% RSLogix 500 project 4P4_E_with_comments.RSS, saved by version 8.30.00.16 %
PROJECT "4P4_E"    % processor: MicroLogix 1000 %

PROGRAM FILES
  LAD 2 "MAIN_PROG"  6 rungs
  LAD 3 "USER_FAULT"  2 rungs
  LAD 4 "HSC_INT"  1 rungs
  LAD 5 "STI_INT"  9 rungs
  LAD 7   40 rungs
  LAD 6, 8, 9, 10, 11, 12, 13, 14, 15, 16: only END

DATA FILES
  O0 OUTPUT  1 elements
  I1 INPUT  2 elements
  S2 STATUS  33 elements
  B3 BINARY  32 elements
  T4 TIMER  40 elements
  C5 COUNTER  32 elements
  R6 CONTROL  16 elements
  N7 INTEGER  105 elements

LADDER 2 "MAIN_PROG"
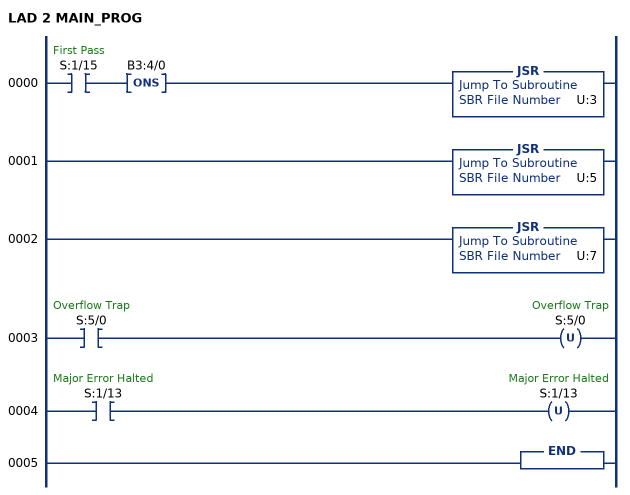
% Rung: 0 %
SOR XIC S:1/15 OSR B3:4/0 JSR U:3 EOR
%   S:1/15  "First Pass" %
% Rung: 1 %
SOR JSR U:5 EOR
% Rung: 2 %
SOR JSR U:7 EOR
% Rung: 3 %
SOR XIC S:5/0 OTU S:5/0 EOR
%   S:5/0  "Overflow Trap" %
% Rung: 4 %
SOR XIC S:1/13 OTU S:1/13 EOR
%   S:1/13  "Major Error Halted" %
% Rung: 5 %
SOR END EOR

LADDER 3 "USER_FAULT"
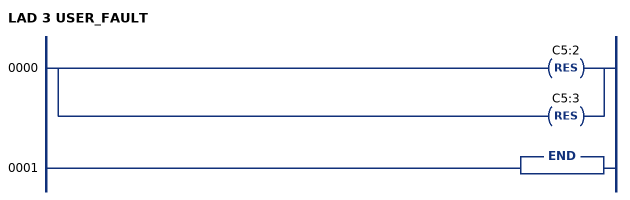
% Rung: 0 %
SOR BST RES C5:2 NXB RES C5:3 BND EOR
% Rung: 1 %
SOR END EOR

LADDER 5 "STI_INT"
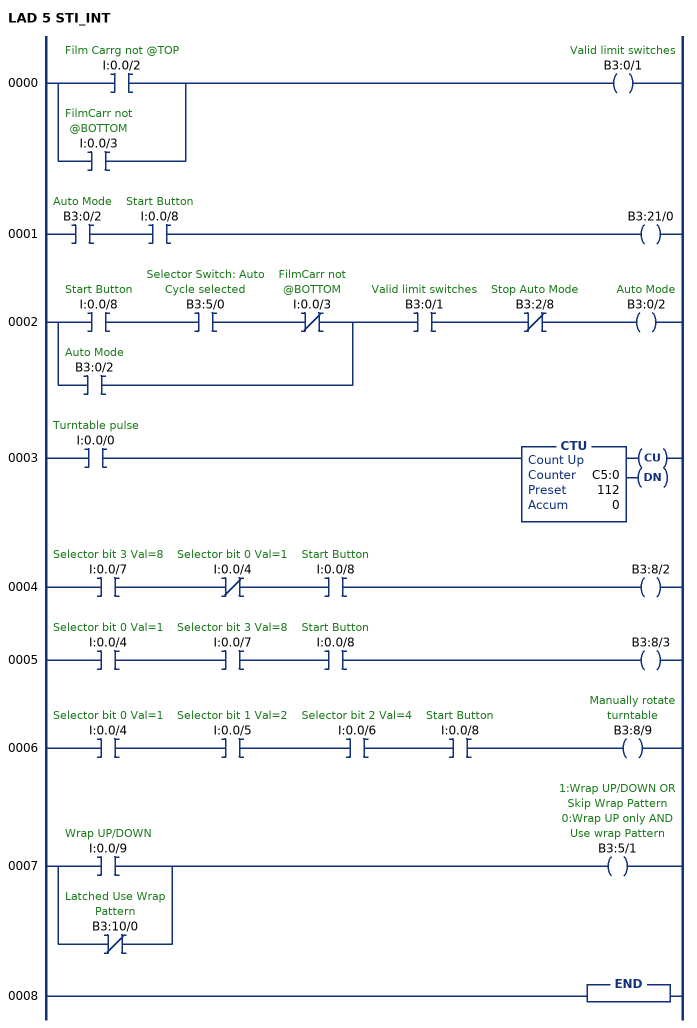
% Rung: 0 %
SOR BST XIC I:0.0/2 NXB XIC I:0.0/3 BND OTE B3:0/1 EOR
%   I:0.0/2  "Film Carrg not @TOP" %
%   XIC I:0.0/2  "1:Film Carr not @TOP" %
%   I:0.0/3  "FilmCarr not @BOTTOM" %
%   XIC I:0.0/3  "1:FilmCarr not@BOTTM" %
%   B3:0/1  "Valid limit switches" %
% Rung: 1 %
SOR XIC B3:0/2 XIC I:0.0/8 OTE B3:21/0 EOR
%   B3:0/2  "Auto Mode" %
%   XIC B3:0/2  "1:Auto" %
%   I:0.0/8  "Start Button" %
% Rung: 2 %
SOR BST XIC I:0.0/8 XIC B3:5/0 XIO I:0.0/3 NXB XIC B3:0/2 BND XIC B3:0/1 XIO B3:2/8 OTE B3:0/2 EOR
%   I:0.0/8  "Start Button" %
%   B3:5/0  "Selector Switch: Auto Cycle selected" %
%   I:0.0/3  "FilmCarr not @BOTTOM" %
%   XIO I:0.0/3  "0:Film Carrg @BOTTOM" %
%   B3:0/2  "Auto Mode" %
%   XIC B3:0/2  "1:Auto" %
%   B3:0/1  "Valid limit switches" %
%   B3:2/8  "Stop Auto Mode" %
%   XIO B3:2/8  "0:Continue Auto Mode" %
% Rung: 3 %
SOR XIC I:0.0/0 CTU C5:0 112 0 EOR
%   I:0.0/0  "Turntable pulse" %
%   XIC I:0.0/0  "1:Turntable pulse on" %
% Rung: 4 %
SOR XIC I:0.0/7 XIO I:0.0/4 XIC I:0.0/8 OTE B3:8/2 EOR
%   I:0.0/7  "Selector bit 3 Val=8" %
%   I:0.0/4  "Selector bit 0 Val=1" %
%   I:0.0/8  "Start Button" %
% Rung: 5 %
SOR XIC I:0.0/4 XIC I:0.0/7 XIC I:0.0/8 OTE B3:8/3 EOR
%   I:0.0/4  "Selector bit 0 Val=1" %
%   I:0.0/7  "Selector bit 3 Val=8" %
%   I:0.0/8  "Start Button" %
% Rung: 6 %
SOR XIC I:0.0/4 XIC I:0.0/5 XIC I:0.0/6 XIC I:0.0/8 OTE B3:8/9 EOR
%   I:0.0/4  "Selector bit 0 Val=1" %
%   I:0.0/5  "Selector bit 1 Val=2" %
%   I:0.0/6  "Selector bit 2 Val=4" %
%   I:0.0/8  "Start Button" %
%   B3:8/9  "Manually rotate turntable" %
% Rung: 7 %
SOR BST XIC I:0.0/9 NXB XIO B3:10/0 BND OTE B3:5/1 EOR
%   I:0.0/9  "Wrap UP/DOWN" %
%   B3:10/0  "Latched Use Wrap Pattern" %
%   XIO B3:10/0  "0:Skip Wrap Pattern" %
%   B3:5/1  "1:Wrap UP/DOWN OR Skip Wrap Pattern 0:Wrap UP only AND Use wrap Pattern" %
% Rung: 8 %
SOR END EOR

LADDER 7
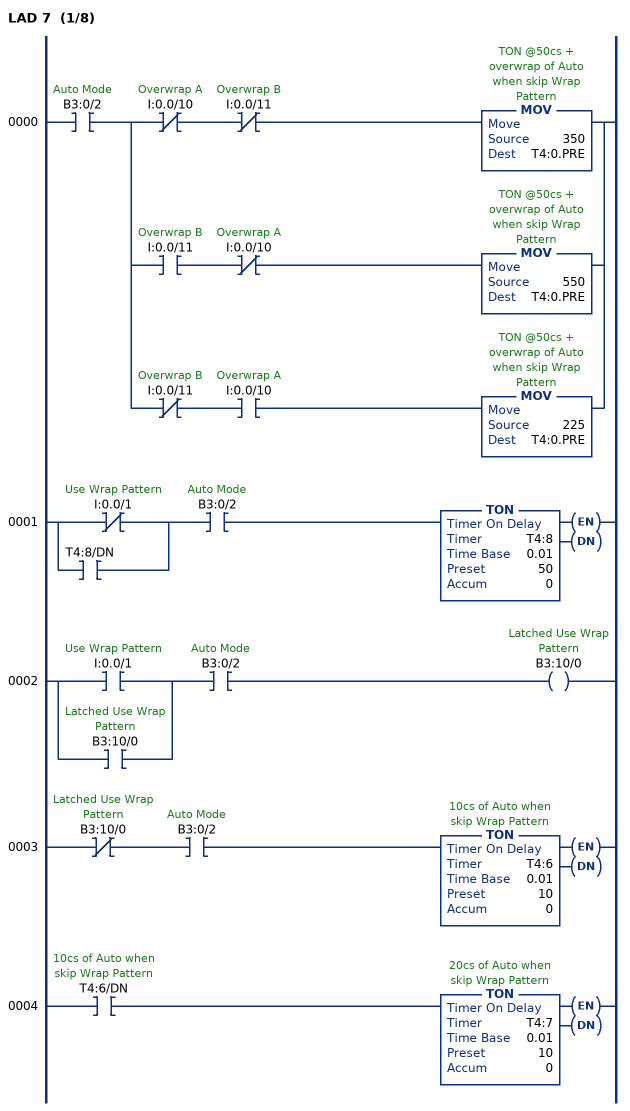
% Rung: 0 %
SOR XIC B3:0/2 BST XIO I:0.0/10 XIO I:0.0/11 MOV 350 T4:0.PRE NXB XIC I:0.0/11 XIO I:0.0/10 MOV 550 T4:0.PRE NXB XIO I:0.0/11 XIC I:0.0/10 MOV 225 T4:0.PRE BND EOR
%   B3:0/2  "Auto Mode" %
%   XIC B3:0/2  "1:Auto" %
%   I:0.0/10  "Overwrap A" %
%   I:0.0/11  "Overwrap B" %
%   T4:0  "TON @50cs + overwrap of Auto when skip Wrap Pattern" %
% Rung: 1 %
SOR BST XIO I:0.0/1 NXB XIC T4:8/DN BND XIC B3:0/2 TON T4:8 0.01 50 0 EOR
%   I:0.0/1  "Use Wrap Pattern" %
%   XIO I:0.0/1  "0:Skip Wrap Pattern => No UP/DOWN" %
%   B3:0/2  "Auto Mode" %
%   XIC B3:0/2  "1:Auto" %
% Rung: 2 %
SOR BST XIC I:0.0/1 NXB XIC B3:10/0 BND XIC B3:0/2 OTE B3:10/0 EOR
%   I:0.0/1  "Use Wrap Pattern" %
%   XIC I:0.0/1  "1:Use Wrap Pattern" %
%   B3:10/0  "Latched Use Wrap Pattern" %
%   B3:0/2  "Auto Mode" %
%   XIC B3:0/2  "1:Auto" %
% Rung: 3 %
SOR XIO B3:10/0 XIC B3:0/2 TON T4:6 0.01 10 0 EOR
%   B3:10/0  "Latched Use Wrap Pattern" %
%   XIO B3:10/0  "0:Skip Wrap Pattern" %
%   B3:0/2  "Auto Mode" %
%   XIC B3:0/2  "1:Auto" %
%   T4:6  "10cs of Auto when skip Wrap Pattern" %
% Rung: 4 %
SOR XIC T4:6/DN TON T4:7 0.01 10 0 EOR
%   T4:6  "10cs of Auto when skip Wrap Pattern" %
%   XIC T4:6/DN  "1:Bypass TOP band 1:10cs+ of Auto when skip Wrap Pattern" %
%   T4:7  "20cs of Auto when skip Wrap Pattern" %

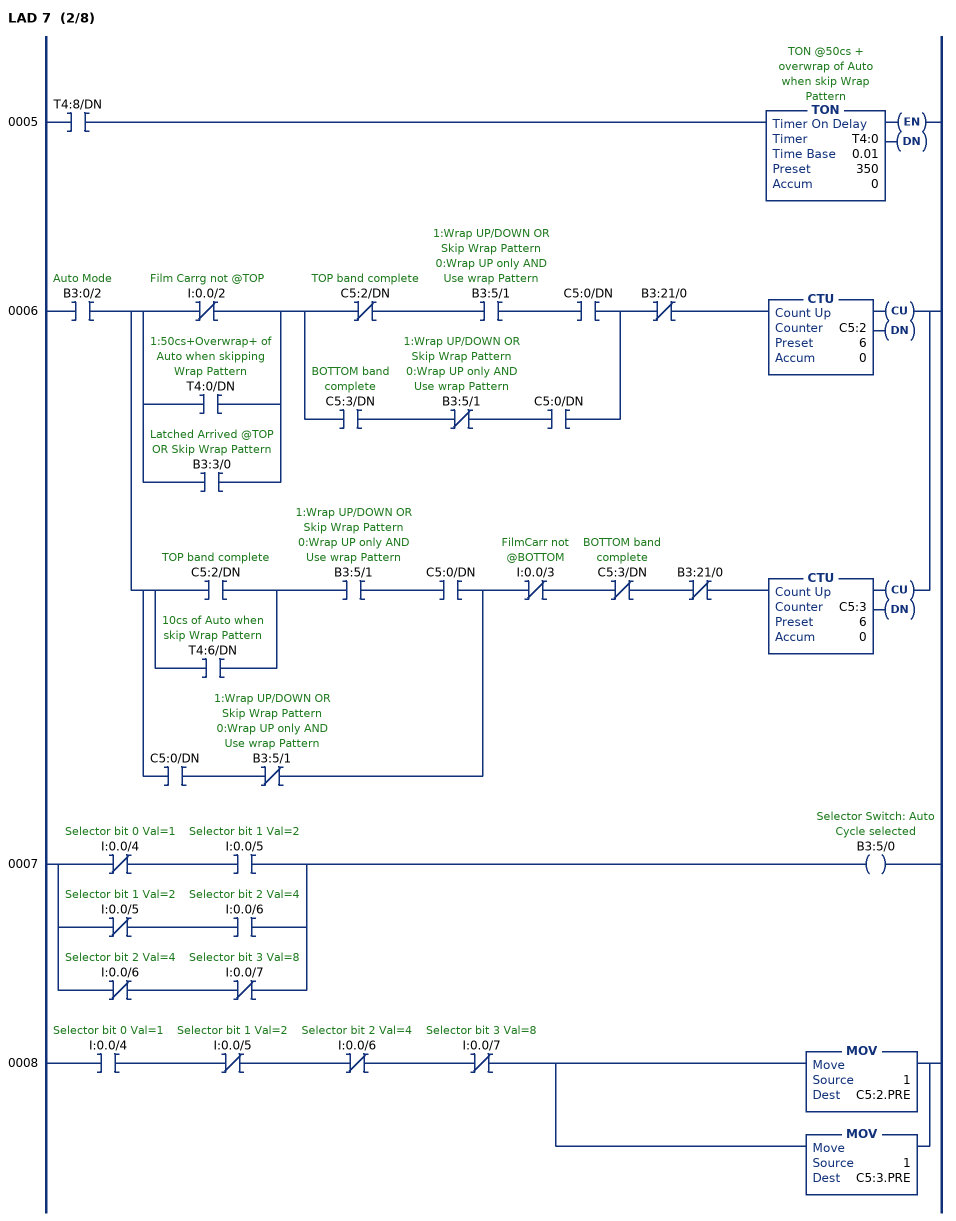
% Rung: 5 %
SOR XIC T4:8/DN TON T4:0 0.01 350 0 EOR
%   T4:0  "TON @50cs + overwrap of Auto when skip Wrap Pattern" %
% Rung: 6 %
SOR XIC B3:0/2 BST BST XIO I:0.0/2 NXB XIC T4:0/DN NXB XIC B3:3/0 BND BST XIO C5:2/DN XIC B3:5/1 XIC C5:0/DN NXB XIC C5:3/DN XIO B3:5/1 XIC C5:0/DN BND XIO B3:21/0 CTU C5:2 6 0 NXB BST BST XIC C5:2/DN NXB XIC T4:6/DN BND XIC B3:5/1 XIC C5:0/DN NXB XIC C5:0/DN XIO B3:5/1 BND XIO I:0.0/3 XIO C5:3/DN XIO B3:21/0 CTU C5:3 6 0 BND EOR
%   B3:0/2  "Auto Mode" %
%   XIC B3:0/2  "1:Auto" %
%   I:0.0/2  "Film Carrg not @TOP" %
%   XIO I:0.0/2  "0:Film Carriage @TOP" %
%   T4:0/DN  "1:50cs+Overwrap+ of Auto when skipping Wrap Pattern" %
%   B3:3/0  "Latched Arrived @TOP OR Skip Wrap Pattern" %
%   XIC B3:3/0  "1:Arrived @TOP OR Skip Wrap Pattern" %
%   C5:2/DN  "TOP band complete" %
%   B3:5/1  "1:Wrap UP/DOWN OR Skip Wrap Pattern 0:Wrap UP only AND Use wrap Pattern" %
%   XIC B3:5/1  "1:Bypass BOTTOM band 1:Wrap UP/DOWN OR Skip Wrap Pattern" %
%   C5:3/DN  "BOTTOM band complete" %
%   XIO B3:5/1  "0:Wrap UP only AND Use wrap Pattern" %
%   T4:6  "10cs of Auto when skip Wrap Pattern" %
%   XIC T4:6/DN  "1:Bypass TOP band 1:10cs+ of Auto when skip Wrap Pattern" %
%   I:0.0/3  "FilmCarr not @BOTTOM" %
%   XIO I:0.0/3  "0:Film Carrg @BOTTOM" %
% Rung: 7 %
SOR BST XIO I:0.0/4 XIC I:0.0/5 NXB XIO I:0.0/5 XIC I:0.0/6 NXB XIO I:0.0/6 XIO I:0.0/7 BND OTE B3:5/0 EOR
%   I:0.0/4  "Selector bit 0 Val=1" %
%   I:0.0/5  "Selector bit 1 Val=2" %
%   I:0.0/6  "Selector bit 2 Val=4" %
%   I:0.0/7  "Selector bit 3 Val=8" %
%   B3:5/0  "Selector Switch: Auto Cycle selected" %
% Rung: 8 %
SOR XIC I:0.0/4 XIO I:0.0/5 XIO I:0.0/6 XIO I:0.0/7 BST MOV 1 C5:2.PRE NXB MOV 1 C5:3.PRE BND EOR
%   I:0.0/4  "Selector bit 0 Val=1" %
%   I:0.0/5  "Selector bit 1 Val=2" %
%   I:0.0/6  "Selector bit 2 Val=4" %
%   I:0.0/7  "Selector bit 3 Val=8" %

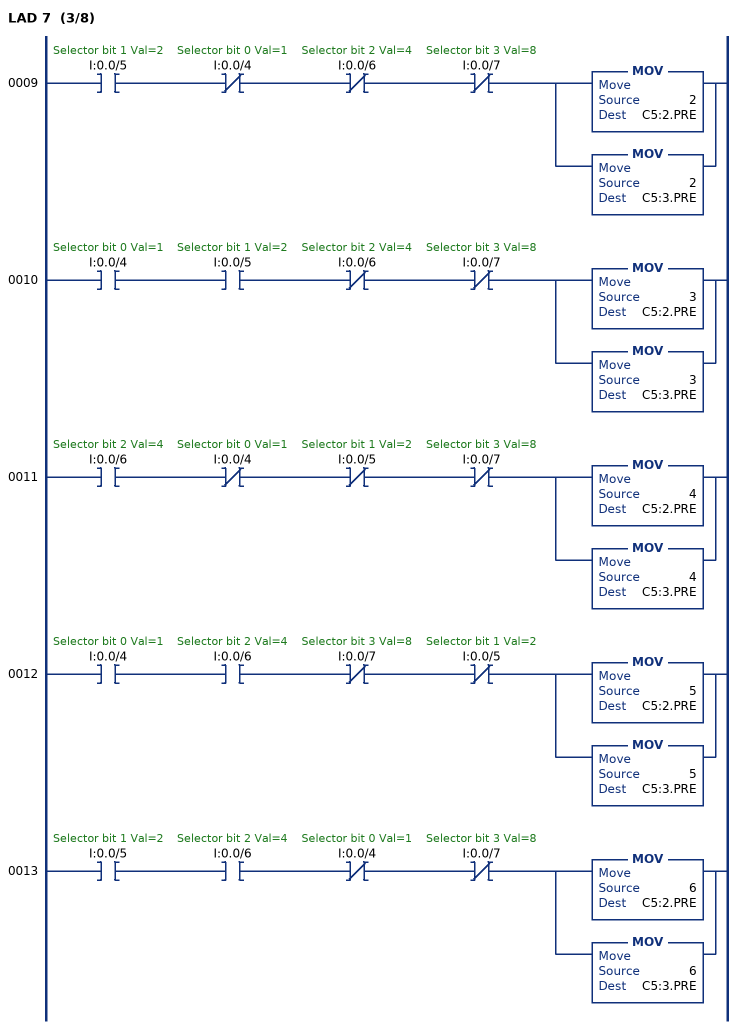
% Rung: 9 %
SOR XIC I:0.0/5 XIO I:0.0/4 XIO I:0.0/6 XIO I:0.0/7 BST MOV 2 C5:2.PRE NXB MOV 2 C5:3.PRE BND EOR
%   I:0.0/5  "Selector bit 1 Val=2" %
%   I:0.0/4  "Selector bit 0 Val=1" %
%   I:0.0/6  "Selector bit 2 Val=4" %
%   I:0.0/7  "Selector bit 3 Val=8" %
% Rung: 10 %
SOR XIC I:0.0/4 XIC I:0.0/5 XIO I:0.0/6 XIO I:0.0/7 BST MOV 3 C5:2.PRE NXB MOV 3 C5:3.PRE BND EOR
%   I:0.0/4  "Selector bit 0 Val=1" %
%   I:0.0/5  "Selector bit 1 Val=2" %
%   I:0.0/6  "Selector bit 2 Val=4" %
%   I:0.0/7  "Selector bit 3 Val=8" %
% Rung: 11 %
SOR XIC I:0.0/6 XIO I:0.0/4 XIO I:0.0/5 XIO I:0.0/7 BST MOV 4 C5:2.PRE NXB MOV 4 C5:3.PRE BND EOR
%   I:0.0/6  "Selector bit 2 Val=4" %
%   I:0.0/4  "Selector bit 0 Val=1" %
%   I:0.0/5  "Selector bit 1 Val=2" %
%   I:0.0/7  "Selector bit 3 Val=8" %
% Rung: 12 %
SOR XIC I:0.0/4 XIC I:0.0/6 XIO I:0.0/7 XIO I:0.0/5 BST MOV 5 C5:2.PRE NXB MOV 5 C5:3.PRE BND EOR
%   I:0.0/4  "Selector bit 0 Val=1" %
%   I:0.0/6  "Selector bit 2 Val=4" %
%   I:0.0/7  "Selector bit 3 Val=8" %
%   I:0.0/5  "Selector bit 1 Val=2" %
% Rung: 13 %
SOR XIC I:0.0/5 XIC I:0.0/6 XIO I:0.0/4 XIO I:0.0/7 BST MOV 6 C5:2.PRE NXB MOV 6 C5:3.PRE BND EOR
%   I:0.0/5  "Selector bit 1 Val=2" %
%   I:0.0/6  "Selector bit 2 Val=4" %
%   I:0.0/4  "Selector bit 0 Val=1" %
%   I:0.0/7  "Selector bit 3 Val=8" %

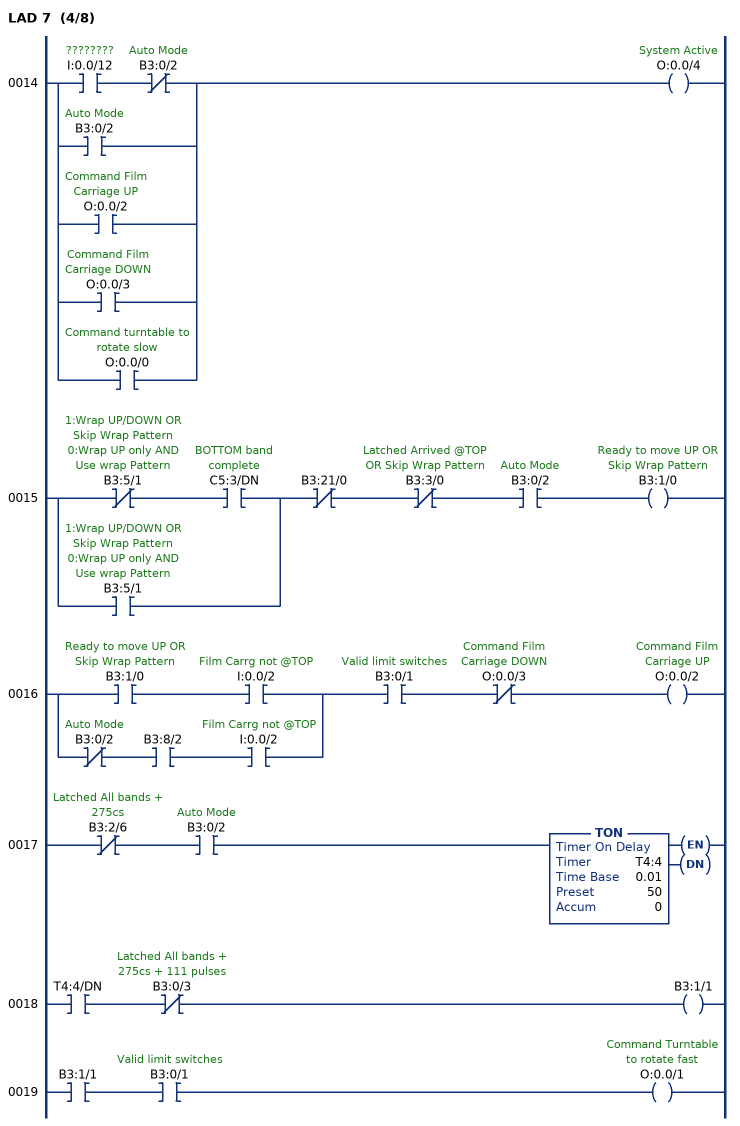
% Rung: 14 %
SOR BST XIC I:0.0/12 XIO B3:0/2 NXB XIC B3:0/2 NXB XIC O:0.0/2 NXB XIC O:0.0/3 NXB XIC O:0.0/0 BND OTE O:0.0/4 EOR
%   I:0.0/12  "????????" %
%   B3:0/2  "Auto Mode" %
%   XIO B3:0/2  "0:Manual" %
%   XIC B3:0/2  "1:Auto" %
%   O:0.0/2  "Command Film Carriage UP" %
%   O:0.0/3  "Command Film Carriage DOWN" %
%   O:0.0/0  "Command turntable to rotate slow" %
%   O:0.0/4  "System Active" %
% Rung: 15 %
SOR BST XIO B3:5/1 XIC C5:3/DN NXB XIC B3:5/1 BND XIO B3:21/0 XIO B3:3/0 XIC B3:0/2 OTE B3:1/0 EOR
%   B3:5/1  "1:Wrap UP/DOWN OR Skip Wrap Pattern 0:Wrap UP only AND Use wrap Pattern" %
%   XIO B3:5/1  "0:Wrap UP only AND Use wrap Pattern" %
%   C5:3/DN  "BOTTOM band complete" %
%   XIC B3:5/1  "1:Bypass BOTTOM band 1:Wrap UP/DOWN OR Skip Wrap Pattern" %
%   B3:3/0  "Latched Arrived @TOP OR Skip Wrap Pattern" %
%   XIO B3:3/0  "0:NOT arrived @TOP AND Use Wrap Pattern" %
%   B3:0/2  "Auto Mode" %
%   XIC B3:0/2  "1:Auto" %
%   B3:1/0  "Ready to move UP OR Skip Wrap Pattern" %
% Rung: 16 %
SOR BST XIC B3:1/0 XIC I:0.0/2 NXB XIO B3:0/2 XIC B3:8/2 XIC I:0.0/2 BND XIC B3:0/1 XIO O:0.0/3 OTE O:0.0/2 EOR
%   B3:1/0  "Ready to move UP OR Skip Wrap Pattern" %
%   I:0.0/2  "Film Carrg not @TOP" %
%   XIC I:0.0/2  "1:Film Carr not @TOP" %
%   B3:0/2  "Auto Mode" %
%   XIO B3:0/2  "0:Manual" %
%   B3:0/1  "Valid limit switches" %
%   O:0.0/3  "Command Film Carriage DOWN" %
%   O:0.0/2  "Command Film Carriage UP" %
% Rung: 17 %
SOR XIO B3:2/6 XIC B3:0/2 TON T4:4 0.01 50 0 EOR
%   B3:2/6  "Latched All bands + 275cs" %
%   XIO B3:2/6  "Not yet 275cs past all bands complete" %
%   B3:0/2  "Auto Mode" %
%   XIC B3:0/2  "1:Auto" %
% Rung: 18 %
SOR XIC T4:4/DN XIO B3:0/3 OTE B3:1/1 EOR
%   B3:0/3  "Latched All bands + 275cs + 111 pulses" %
%   XIO B3:0/3  "0:Not done wrapping" %
% Rung: 19 %
SOR XIC B3:1/1 XIC B3:0/1 OTE O:0.0/1 EOR
%   B3:0/1  "Valid limit switches" %
%   O:0.0/1  "Command Turntable to rotate fast" %

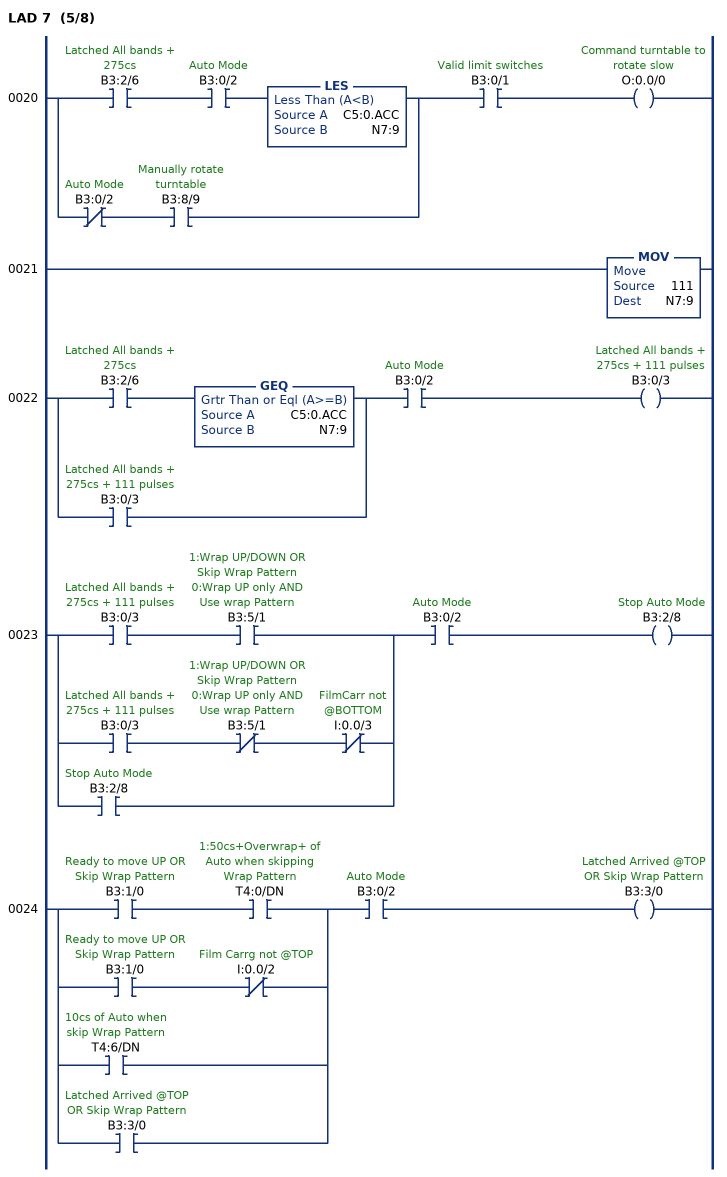
% Rung: 20 %
SOR BST XIC B3:2/6 XIC B3:0/2 LES C5:0.ACC N7:9 NXB XIO B3:0/2 XIC B3:8/9 BND XIC B3:0/1 OTE O:0.0/0 EOR
%   B3:2/6  "Latched All bands + 275cs" %
%   XIC B3:2/6  "1:All bands + 275cs" %
%   B3:0/2  "Auto Mode" %
%   XIC B3:0/2  "1:Auto" %
%   XIO B3:0/2  "0:Manual" %
%   B3:8/9  "Manually rotate turntable" %
%   B3:0/1  "Valid limit switches" %
%   O:0.0/0  "Command turntable to rotate slow" %
% Rung: 21 %
SOR MOV 111 N7:9 EOR
% Rung: 22 %
SOR BST XIC B3:2/6 GEQ C5:0.ACC N7:9 NXB XIC B3:0/3 BND XIC B3:0/2 OTE B3:0/3 EOR
%   B3:2/6  "Latched All bands + 275cs" %
%   XIC B3:2/6  "1:All bands + 275cs" %
%   B3:0/3  "Latched All bands + 275cs + 111 pulses" %
%   XIC B3:0/3  "1:Done wrapping" %
%   B3:0/2  "Auto Mode" %
%   XIC B3:0/2  "1:Auto" %
% Rung: 23 %
SOR BST BST XIC B3:0/3 XIC B3:5/1 NXB XIC B3:0/3 XIO B3:5/1 XIO I:0.0/3 BND NXB XIC B3:2/8 BND XIC B3:0/2 OTE B3:2/8 EOR
%   B3:0/3  "Latched All bands + 275cs + 111 pulses" %
%   XIC B3:0/3  "1:Done wrapping" %
%   B3:5/1  "1:Wrap UP/DOWN OR Skip Wrap Pattern 0:Wrap UP only AND Use wrap Pattern" %
%   XIC B3:5/1  "1:Bypass BOTTOM band 1:Wrap UP/DOWN OR Skip Wrap Pattern" %
%   XIO B3:5/1  "0:Wrap UP only AND Use wrap Pattern" %
%   I:0.0/3  "FilmCarr not @BOTTOM" %
%   XIO I:0.0/3  "0:Film Carrg @BOTTOM" %
%   B3:2/8  "Stop Auto Mode" %
%   XIC B3:2/8  "1:Stop Auto Mode" %
%   B3:0/2  "Auto Mode" %
%   XIC B3:0/2  "1:Auto" %
% Rung: 24 %
SOR BST XIC B3:1/0 XIC T4:0/DN NXB XIC B3:1/0 XIO I:0.0/2 NXB XIC T4:6/DN NXB XIC B3:3/0 BND XIC B3:0/2 OTE B3:3/0 EOR
%   B3:1/0  "Ready to move UP OR Skip Wrap Pattern" %
%   T4:0/DN  "1:50cs+Overwrap+ of Auto when skipping Wrap Pattern" %
%   I:0.0/2  "Film Carrg not @TOP" %
%   XIO I:0.0/2  "0:Film Carriage @TOP" %
%   T4:6  "10cs of Auto when skip Wrap Pattern" %
%   XIC T4:6/DN  "1:Bypass TOP band 1:10cs+ of Auto when skip Wrap Pattern" %
%   B3:3/0  "Latched Arrived @TOP OR Skip Wrap Pattern" %
%   XIC B3:3/0  "1:Arrived @TOP OR Skip Wrap Pattern" %
%   B3:0/2  "Auto Mode" %
%   XIC B3:0/2  "1:Auto" %

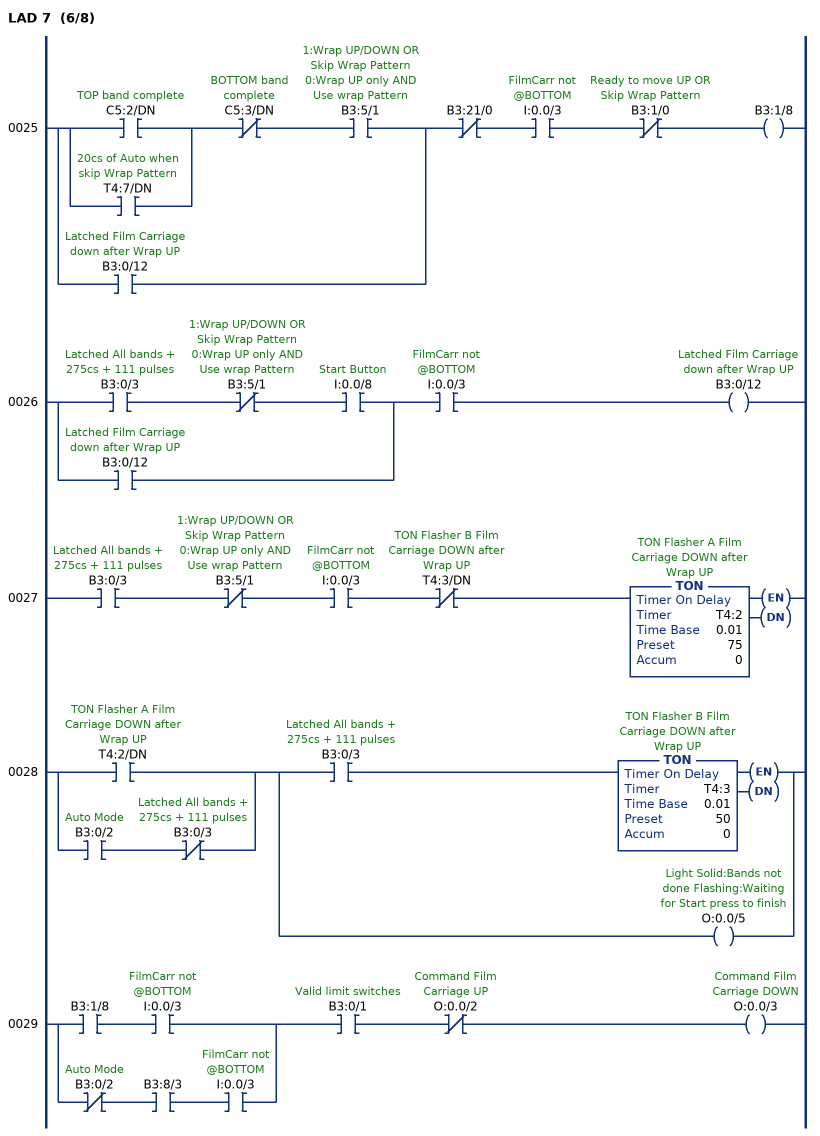
% Rung: 25 %
SOR BST BST XIC C5:2/DN NXB XIC T4:7/DN BND XIO C5:3/DN XIC B3:5/1 NXB XIC B3:0/12 BND XIO B3:21/0 XIC I:0.0/3 XIO B3:1/0 OTE B3:1/8 EOR
%   C5:2/DN  "TOP band complete" %
%   T4:7  "20cs of Auto when skip Wrap Pattern" %
%   XIC T4:7/DN  "1:Bypass TOP band 1:20cs+ of Auto when skip Wrap Pattern" %
%   C5:3/DN  "BOTTOM band complete" %
%   B3:5/1  "1:Wrap UP/DOWN OR Skip Wrap Pattern 0:Wrap UP only AND Use wrap Pattern" %
%   XIC B3:5/1  "1:Bypass BOTTOM band 1:Wrap UP/DOWN OR Skip Wrap Pattern" %
%   B3:0/12  "Latched Film Carriage down after Wrap UP" %
%   XIC B3:0/12  "1:Film Carriage DOWN after Wrap UP" %
%   I:0.0/3  "FilmCarr not @BOTTOM" %
%   XIC I:0.0/3  "1:FilmCarr not@BOTTM" %
%   B3:1/0  "Ready to move UP OR Skip Wrap Pattern" %
% Rung: 26 %
SOR BST XIC B3:0/3 XIO B3:5/1 XIC I:0.0/8 NXB XIC B3:0/12 BND XIC I:0.0/3 OTE B3:0/12 EOR
%   B3:0/3  "Latched All bands + 275cs + 111 pulses" %
%   XIC B3:0/3  "1:Done wrapping" %
%   B3:5/1  "1:Wrap UP/DOWN OR Skip Wrap Pattern 0:Wrap UP only AND Use wrap Pattern" %
%   XIO B3:5/1  "0:Wrap UP only AND Use wrap Pattern" %
%   I:0.0/8  "Start Button" %
%   B3:0/12  "Latched Film Carriage down after Wrap UP" %
%   XIC B3:0/12  "1:Film Carriage DOWN after Wrap UP" %
%   I:0.0/3  "FilmCarr not @BOTTOM" %
%   XIC I:0.0/3  "1:FilmCarr not@BOTTM" %
% Rung: 27 %
SOR XIC B3:0/3 XIO B3:5/1 XIC I:0.0/3 XIO T4:3/DN TON T4:2 0.01 75 0 EOR
%   B3:0/3  "Latched All bands + 275cs + 111 pulses" %
%   XIC B3:0/3  "1:Done wrapping" %
%   B3:5/1  "1:Wrap UP/DOWN OR Skip Wrap Pattern 0:Wrap UP only AND Use wrap Pattern" %
%   XIO B3:5/1  "0:Wrap UP only AND Use wrap Pattern" %
%   I:0.0/3  "FilmCarr not @BOTTOM" %
%   XIC I:0.0/3  "1:FilmCarr not@BOTTM" %
%   T4:3  "TON Flasher B Film Carriage DOWN after Wrap UP" %
%   T4:2  "TON Flasher A Film Carriage DOWN after Wrap UP" %
% Rung: 28 %
SOR BST XIC T4:2/DN NXB XIC B3:0/2 XIO B3:0/3 BND BST XIC B3:0/3 TON T4:3 0.01 50 0 NXB OTE O:0.0/5 BND EOR
%   T4:2  "TON Flasher A Film Carriage DOWN after Wrap UP" %
%   B3:0/2  "Auto Mode" %
%   XIC B3:0/2  "1:Auto" %
%   B3:0/3  "Latched All bands + 275cs + 111 pulses" %
%   XIO B3:0/3  "0:Not done wrapping" %
%   XIC B3:0/3  "1:Done wrapping" %
%   T4:3  "TON Flasher B Film Carriage DOWN after Wrap UP" %
%   O:0.0/5  "Light Solid:Bands not done Flashing:Waiting for Start press to finish" %
% Rung: 29 %
SOR BST XIC B3:1/8 XIC I:0.0/3 NXB XIO B3:0/2 XIC B3:8/3 XIC I:0.0/3 BND XIC B3:0/1 XIO O:0.0/2 OTE O:0.0/3 EOR
%   I:0.0/3  "FilmCarr not @BOTTOM" %
%   XIC I:0.0/3  "1:FilmCarr not@BOTTM" %
%   B3:0/2  "Auto Mode" %
%   XIO B3:0/2  "0:Manual" %
%   B3:0/1  "Valid limit switches" %
%   O:0.0/2  "Command Film Carriage UP" %
%   O:0.0/3  "Command Film Carriage DOWN" %

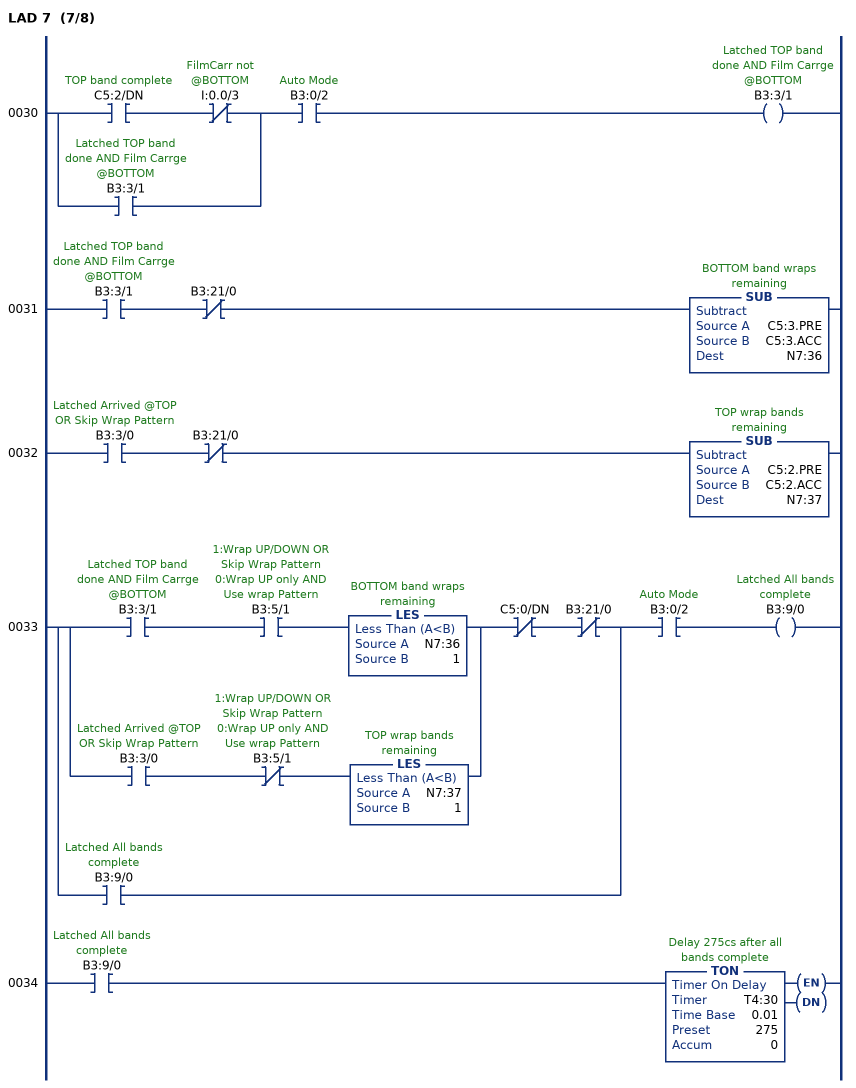
% Rung: 30 %
SOR BST XIC C5:2/DN XIO I:0.0/3 NXB XIC B3:3/1 BND XIC B3:0/2 OTE B3:3/1 EOR
%   C5:2/DN  "TOP band complete" %
%   I:0.0/3  "FilmCarr not @BOTTOM" %
%   XIO I:0.0/3  "0:Film Carrg @BOTTOM" %
%   B3:3/1  "Latched TOP band done AND Film Carrge @BOTTOM" %
%   B3:0/2  "Auto Mode" %
%   XIC B3:0/2  "1:Auto" %
% Rung: 31 %
SOR XIC B3:3/1 XIO B3:21/0 SUB C5:3.PRE C5:3.ACC N7:36 EOR
%   B3:3/1  "Latched TOP band done AND Film Carrge @BOTTOM" %
%   N7:36  "BOTTOM band wraps remaining" %
% Rung: 32 %
SOR XIC B3:3/0 XIO B3:21/0 SUB C5:2.PRE C5:2.ACC N7:37 EOR
%   B3:3/0  "Latched Arrived @TOP OR Skip Wrap Pattern" %
%   XIC B3:3/0  "1:Arrived @TOP OR Skip Wrap Pattern" %
%   N7:37  "TOP wrap bands remaining" %
% Rung: 33 %
SOR BST BST XIC B3:3/1 XIC B3:5/1 LES N7:36 1 NXB XIC B3:3/0 XIO B3:5/1 LES N7:37 1 BND XIO C5:0/DN XIO B3:21/0 NXB XIC B3:9/0 BND XIC B3:0/2 OTE B3:9/0 EOR
%   B3:3/1  "Latched TOP band done AND Film Carrge @BOTTOM" %
%   B3:5/1  "1:Wrap UP/DOWN OR Skip Wrap Pattern 0:Wrap UP only AND Use wrap Pattern" %
%   XIC B3:5/1  "1:Bypass BOTTOM band 1:Wrap UP/DOWN OR Skip Wrap Pattern" %
%   N7:36  "BOTTOM band wraps remaining" %
%   B3:3/0  "Latched Arrived @TOP OR Skip Wrap Pattern" %
%   XIC B3:3/0  "1:Arrived @TOP OR Skip Wrap Pattern" %
%   XIO B3:5/1  "0:Wrap UP only AND Use wrap Pattern" %
%   N7:37  "TOP wrap bands remaining" %
%   B3:9/0  "Latched All bands complete" %
%   B3:0/2  "Auto Mode" %
%   XIC B3:0/2  "1:Auto" %
% Rung: 34 %
SOR XIC B3:9/0 TON T4:30 0.01 275 0 EOR
%   B3:9/0  "Latched All bands complete" %
%   T4:30  "Delay 275cs after all bands complete" %

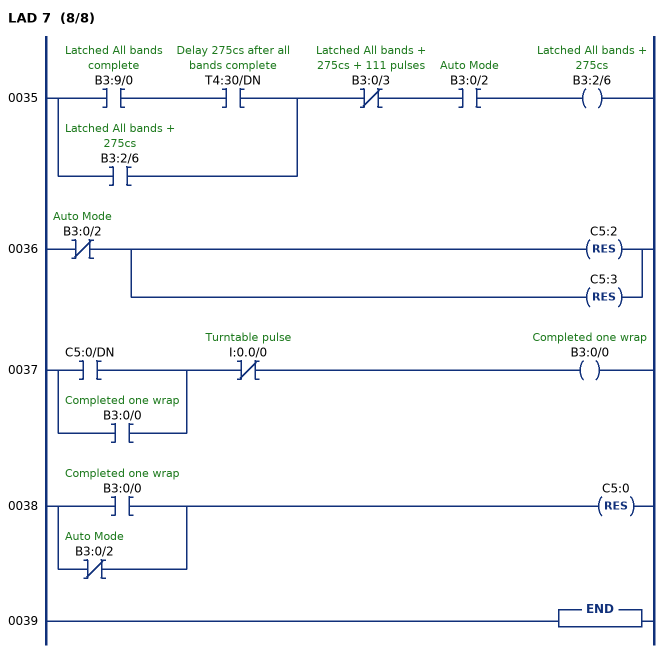
% Rung: 35 %
SOR BST XIC B3:9/0 XIC T4:30/DN NXB XIC B3:2/6 BND XIO B3:0/3 XIC B3:0/2 OTE B3:2/6 EOR
%   B3:9/0  "Latched All bands complete" %
%   T4:30  "Delay 275cs after all bands complete" %
%   XIC T4:30/DN  "1:All bands + 275cs+" %
%   B3:2/6  "Latched All bands + 275cs" %
%   XIC B3:2/6  "1:All bands + 275cs" %
%   B3:0/3  "Latched All bands + 275cs + 111 pulses" %
%   XIO B3:0/3  "0:Not done wrapping" %
%   B3:0/2  "Auto Mode" %
%   XIC B3:0/2  "1:Auto" %
% Rung: 36 %
SOR XIO B3:0/2 BST RES C5:2 NXB RES C5:3 BND EOR
%   B3:0/2  "Auto Mode" %
%   XIO B3:0/2  "0:Manual" %
% Rung: 37 %
SOR BST XIC C5:0/DN NXB XIC B3:0/0 BND XIO I:0.0/0 OTE B3:0/0 EOR
%   B3:0/0  "Completed one wrap" %
%   I:0.0/0  "Turntable pulse" %
%   XIO I:0.0/0  "0Turntable pulse off" %
% Rung: 38 %
SOR BST XIC B3:0/0 NXB XIO B3:0/2 BND RES C5:0 EOR
%   B3:0/0  "Completed one wrap" %
%   B3:0/2  "Auto Mode" %
%   XIO B3:0/2  "0:Manual" %
% Rung: 39 %
SOR END EOR

DATA TABLE (non-zero values as saved)
DATA B3
% B3:0 % 0X0070 0X0010 0X0006 0X0104 0X0000 0X0003 0X0010 0X0000 0X0000 0X0000
% B3:10 % 0X040A 0X0040 0X0300 0X0000 0X0000 0X0000 0X0000 0X0000 0X0000 0X0000
% B3:20 % 0X0028 0X0000 0X0000 0X0000 0X0000 0X0000 0X0000 0X0000 0X0000 0X0000
% B3:30 % 0XCC3A 0X0001
DATA T4
% .PRE .ACC %
% T4:0 % 350 0
% T4:1 % 10 0
% T4:2 % 75 0
% T4:3 % 50 0
% T4:4 % 50 0
% T4:6 % 10 0
% T4:7 % 10 0
% T4:8 % 50 0
% T4:9 % 100 0
% T4:11 % 400 0
% T4:12 % 20 0
% T4:13 % 400 400
% T4:14 % 400 0
% T4:15 % 150 150
% T4:16 % 300 300
% T4:17 % 120 0
% T4:18 % 150 0
% T4:19 % 200 0
% T4:20 % 100 0
% T4:21 % 50 0
% T4:22 % 100 0
% T4:23 % 70 0
% T4:24 % 10 0
% T4:25 % 100 0
% T4:26 % 300 0
% T4:27 % 100 0
% T4:29 % 1 1
% T4:30 % 275 0
% T4:31 % 450 0
% T4:32 % 50 50
% T4:34 % 200 0
% T4:36 % 800 0
% T4:37 % 200 0
% T4:38 % 350 0
DATA C5
% .PRE .ACC %
% C5:0 % 112 0
% C5:1 % 9999 1456
% C5:2 % 6 0
% C5:3 % 6 0
% C5:4 % 9999 221
% C5:5 % 9999 0
% C5:6 % 1 0
% C5:7 % 9999 7
% C5:8 % 3 0
% C5:9 % 3 0
% C5:10 % 20 1
% C5:11 % 9999 0
% C5:12 % 9999 2
% C5:14 % 76 0
% C5:15 % 3 0
% C5:16 % 2 1
DATA R6
% .LEN .POS %
% R6:0 % 16 0
DATA N7
% N7:0 % 2 2 2 0 0 0 1 221 112 111
% N7:10 % 80 1 0 0 0 0 0 0 0 0
